PROGRAM MAIN
VAR
	bStartReadRequest 	: BOOL;	
	bStartWriteRequest	: BOOL;
	
	stS7Info			: ST_S7_Info;
	stS7RequestHandling	: ST_S7_RequestHandling;

	(* Read variables *)
	bReadRequestDone	: BOOL;
	stS7Incoming		: ST_S7_Incoming;
	stS7IncomingCyclic	: ST_S7_Incoming_Cyclic;
	
	(* Write variables *)
	bWriteEnable AT%Q*	: BOOL;
	bWriteRequestDone	: BOOL;
	i1write AT%Q*		: INT := 42;
	
	(* State machine variables *)
	nState				: UINT;
	nStateWrite			: UINT;
	
END_VAR

CASE nState OF 
	0: 
		IF bStartReadRequest THEN
			bStartReadRequest := FALSE;
			bReadRequestDone := FALSE;
			nState := nState + 1;
		END_IF

	1:
		stS7RequestHandling.bySendRequest := stS7RequestHandling.byReceiveCounter + 1;
		nState := nState + 1;
		
	2: 
		IF stS7RequestHandling.byReceiveCounter = stS7RequestHandling.bySendRequest THEN
			nState := nState + 1;
		END_IF	
		
	3: 
		bReadRequestDone := TRUE;
		nState := 0;
	
END_CASE

CASE nStateWrite OF
	0:
		IF bStartWriteRequest THEN
			bStartWriteRequest := FALSE;
			bWriteEnable := TRUE;
			nStateWrite := nStateWrite + 1;
		END_IF

	1:
		stS7RequestHandling.bySendRequest := stS7RequestHandling.byReceiveCounter + 1;
		nStateWrite := nStateWrite + 1;
		
	2: 
		IF stS7RequestHandling.byReceiveCounter = stS7RequestHandling.bySendRequest THEN
			bWriteEnable := FALSE;
			nStateWrite := nStateWrite + 1;
		END_IF	
	
	3: 
		bWriteRequestDone := TRUE;
		nStateWrite := 0;
		
END_CASE

END_PROGRAM

(* stored: Version 1.1.0.1, ProductVersion 3.1.4024.4
   POU MAIN: Id {b1e5abb7-541f-47a1-be0f-3c03fc6aac30}, SpecialFunc None *)
